PROGRAM MAIN
VAR
	bS01 : BOOL;
	bS02 : BOOL;
	bQ01 : BOOL;
	bQ02 : BOOL;
END_VAR

bQ01 := (bS01 AND NOT bS02) OR (NOT bS01 AND NOT bS02);
bQ02 := (NOT bS01 AND bS02) OR (NOT bS01 AND NOT bS02);

END_PROGRAM

(* stored: Version 1.1.0.1, ProductVersion 3.1.4024.12
   POU MAIN: Id {db47084a-bd84-46ce-a376-30981b86512a}, SpecialFunc None *)
